(*
Nazwa:			P08_CapFeeder
Opis:			Stacja podajnika nasadek
Wersja:			v0.2
Data:			2024-01-12
Autor:			DP
Urzadzenia:		
Konfiguracja:	
Info:

*)
PROGRAM P08_CapSorter
VAR_INPUT
	IbCapSorterGateScrewerSensor 			:BOOL;			
	IbCapSorterGateWeightSensor				:BOOL;
	//WEJSCIA I WYJSCIA SPRZETOWE
	IbCapSorterDragHomingSensor 			 :BOOL;						// Czujnik bazowania
	QbCapSorterDragActuator               	 :BOOL;						// Siłownikiem przeciągania 
	IbCapSorterDragUpSensor 				 :BOOL;						// Czujnik
	IbCapSorterDragDownSensor 				 :BOOL;						// Czujnik
	                                         
	QbCapSorterDragLeadBefore1Actuator       :BOOL;						// Siłownikiem prowadzenia przed 
	IbCapSorterDragLeadBefore1UpSensor 	 	 :BOOL;						// Czujnik
 	IbCapSorterDragLeadBefore2UpSensor 	 	 :BOOL;						// Czujnik			
	QbCapSorterDragLeadAfter1Actuator        :BOOL;						// Siłownikiem prowadzenia za
	IbCapSorterDragLeadAfter1UpSensor 	 	 :BOOL;						// Czujnik
 	IbCapSorterDragLeadAfter2UpSensor 	 	 :BOOL;						// Czujnik			

END_VAR
VAR
	
	(*******PRZECIAGANIE**********)
	eCapSorterDragStation						: E_Station;
	eCapSorterDragRunningStation				: E_DragStationState;
	fbCapSorterDragState						: FB_State;
	fbCapSorterDragStation						: FB_FormsDragStepper;	
	
	

	
	
	//Pomocnicze
	tofCapSorterDragEnable					: TOF;
	
	//Stoper
	QbCapSorterStoperActuator				: BOOL;				// bit to wysterowania sygnału stopera	
	tpStoperTimerOn							: TP;				// timer do generowania impulsu
	fbStoperSensorDelay						: FB_InputFilter;	// filtr do generowania sygnału 
	lrCapSorterStoperPosition						: LREAL;	
	rtCapSorterStoperDraging: R_TRIG;
	rtCapSorterStoperEndingOfDraging: R_TRIG;	
	//Inne
	bTemp: BOOL;

	rtCapSorterStoperPackMLStarting: R_TRIG;
	bCapSorterStoperWaitingForSensor: BOOL;
	bCapSorterStoperActuatorDelay: BOOL;
	tonbCapSorterStoperActuatorDelay: TON;
	
	//ManualStoper
	rtManualMode	: R_TRIG;
	ftManualMode	: F_TRIG;	
	bCapSorterStoperActuatorLastState	:BOOL;
	
END_VAR

//bCapSorterDisable:=VIS.bCapPuttedCheckIgnoreErrors;


tofCapSorterDragEnable(IN:= GVL.bCapSorterDragEnable, PT:= T#5S);
aLimits();
aStoper();
aDragStation();
aCapSorterWarnings();


(********* GENEROWANIE STANU STACJI DO WIZKI**********)
fbCapSorterDragState(
	eState:=eCapSorterDragStation, 
	bRun:=VIS.bCapSorterDragRun,
	eFormsDragingRunningState:=eCapSorterDragRunningStation, 
	sStateDesc=> VIS.sCapSorterDragState,
	iState=>VIS.iCapSorterDragState);
(***** KONIEC GENEROWANIE STANU STACJI DO WIZKI*******)



IF fbCapSorterDragStation.bCycleDone AND bManualMode THEN
	VIS.bCapSorterDragRun 						:= FALSE;
	GVL.bCapSorterDragPrepareRun				:= FALSE;
END_IF

ACTION aCapSorterWarnings:

//Warning 0
IF stCapSorterRead.eReservedSignals.iReserved20.0 AND NOT CapSorterWarning[0].bWarning THEN
	CapSorterWarning[0].bWarning										:=TRUE;
	CapSorterWarning[0].udiWarningCode									:=41;
	CapSorterWarning[0].sDescription									:='Sorter nasadek | Brak nasadek w zasobniku';
ELSIF NOT stCapSorterRead.eReservedSignals.iReserved20.0 THEN//AND CapSorterWarning[0].bAcknowledge THEN
	CapSorterWarning[0].bWarning										:=FALSE;
	CapSorterWarning[0].bAcknowledge									:=FALSE;
	VIS.uliWarningAcknowledge.27										:=FALSE;
ELSIF CapSorterWarning[0].bAcknowledge THEN                               
	CapSorterWarning[0].bAcknowledge									:=TRUE;
END_IF

//Warning 1
IF stCapSorterRead.eReservedSignals.iReserved20.1 AND NOT CapSorterWarning[1].bWarning THEN
	CapSorterWarning[1].bWarning										:=TRUE;
	CapSorterWarning[1].udiWarningCode									:=42;
	CapSorterWarning[1].sDescription									:='Sorter nasadek | Brak nasadek na stole - sprawdź transporter pośredni';
ELSIF NOT stCapSorterRead.eReservedSignals.iReserved20.1 AND CapSorterWarning[1].bAcknowledge THEN
	CapSorterWarning[1].bWarning										:=FALSE;
	CapSorterWarning[1].bAcknowledge									:=FALSE;
	VIS.uliWarningAcknowledge.28										:=FALSE;
ELSIF CapSorterWarning[1].bAcknowledge THEN
	CapSorterWarning[1].bAcknowledge									:=TRUE;
END_IF

//Warning 2
IF stCapSorterRead.eReservedSignals.iReserved20.2 AND NOT CapSorterWarning[2].bWarning THEN
	CapSorterWarning[2].bWarning										:=TRUE;
	CapSorterWarning[2].udiWarningCode									:=43;
	CapSorterWarning[2].sDescription									:='Sorter nasadek | Niepobrana nasadka przez chwytak 1';
ELSIF NOT stCapSorterRead.eReservedSignals.iReserved20.1 AND CapSorterWarning[2].bAcknowledge THEN
	CapSorterWarning[2].bWarning										:=FALSE;
	CapSorterWarning[2].bAcknowledge									:=FALSE;
	VIS.uliWarningAcknowledge.29										:=FALSE;
ELSIF CapSorterWarning[2].bAcknowledge THEN
	CapSorterWarning[2].bAcknowledge									:=TRUE;
END_IF

//Warning 3
IF stCapSorterRead.eReservedSignals.iReserved20.3 AND NOT CapSorterWarning[3].bWarning THEN
	CapSorterWarning[3].bWarning										:=TRUE;
	CapSorterWarning[3].udiWarningCode									:=44;
	CapSorterWarning[3].sDescription									:='Sorter nasadek | Niepobrana nasadka przez chwytak 2';
ELSIF NOT stCapSorterRead.eReservedSignals.iReserved20.1 AND CapSorterWarning[3].bAcknowledge THEN
	CapSorterWarning[3].bWarning										:=FALSE;
	CapSorterWarning[3].bAcknowledge									:=FALSE;
	VIS.uliWarningAcknowledge.30										:=FALSE;
ELSIF CapSorterWarning[3].bAcknowledge THEN
	CapSorterWarning[3].bAcknowledge									:=TRUE;
END_IF

//Warning 4
IF stCapSorterRead.eReservedSignals.iReserved20.4 AND NOT CapSorterWarning[4].bWarning THEN
	CapSorterWarning[4].bWarning										:=TRUE;
	CapSorterWarning[4].udiWarningCode									:=45;
	CapSorterWarning[4].sDescription									:='Sorter nasadek | Niepobrana nasadka przez chwytak 3';
ELSIF NOT stCapSorterRead.eReservedSignals.iReserved20.1 AND CapSorterWarning[4].bAcknowledge THEN
	CapSorterWarning[4].bWarning										:=FALSE;
	CapSorterWarning[4].bAcknowledge									:=FALSE;
	VIS.uliWarningAcknowledge.31										:=FALSE;
ELSIF CapSorterWarning[4].bAcknowledge THEN
	CapSorterWarning[4].bAcknowledge									:=TRUE;
END_IF

//Warning 5
IF stCapSorterRead.eReservedSignals.iReserved20.5 AND NOT CapSorterWarning[5].bWarning THEN
	CapSorterWarning[5].bWarning										:=TRUE;
	CapSorterWarning[5].udiWarningCode									:=46;
	CapSorterWarning[5].sDescription									:='Sorter nasadek | Niepobrana nasadka przez chwytak 4';	
ELSIF NOT stCapSorterRead.eReservedSignals.iReserved20.1 AND CapSorterWarning[5].bAcknowledge THEN
	CapSorterWarning[5].bWarning										:=FALSE;
	CapSorterWarning[5].bAcknowledge									:=FALSE;
	VIS.uliWarningAcknowledge.32										:=FALSE;
ELSIF CapSorterWarning[5].bAcknowledge THEN
	CapSorterWarning[5].bAcknowledge									:=TRUE;
END_IF
END_ACTION

ACTION aDragStation:
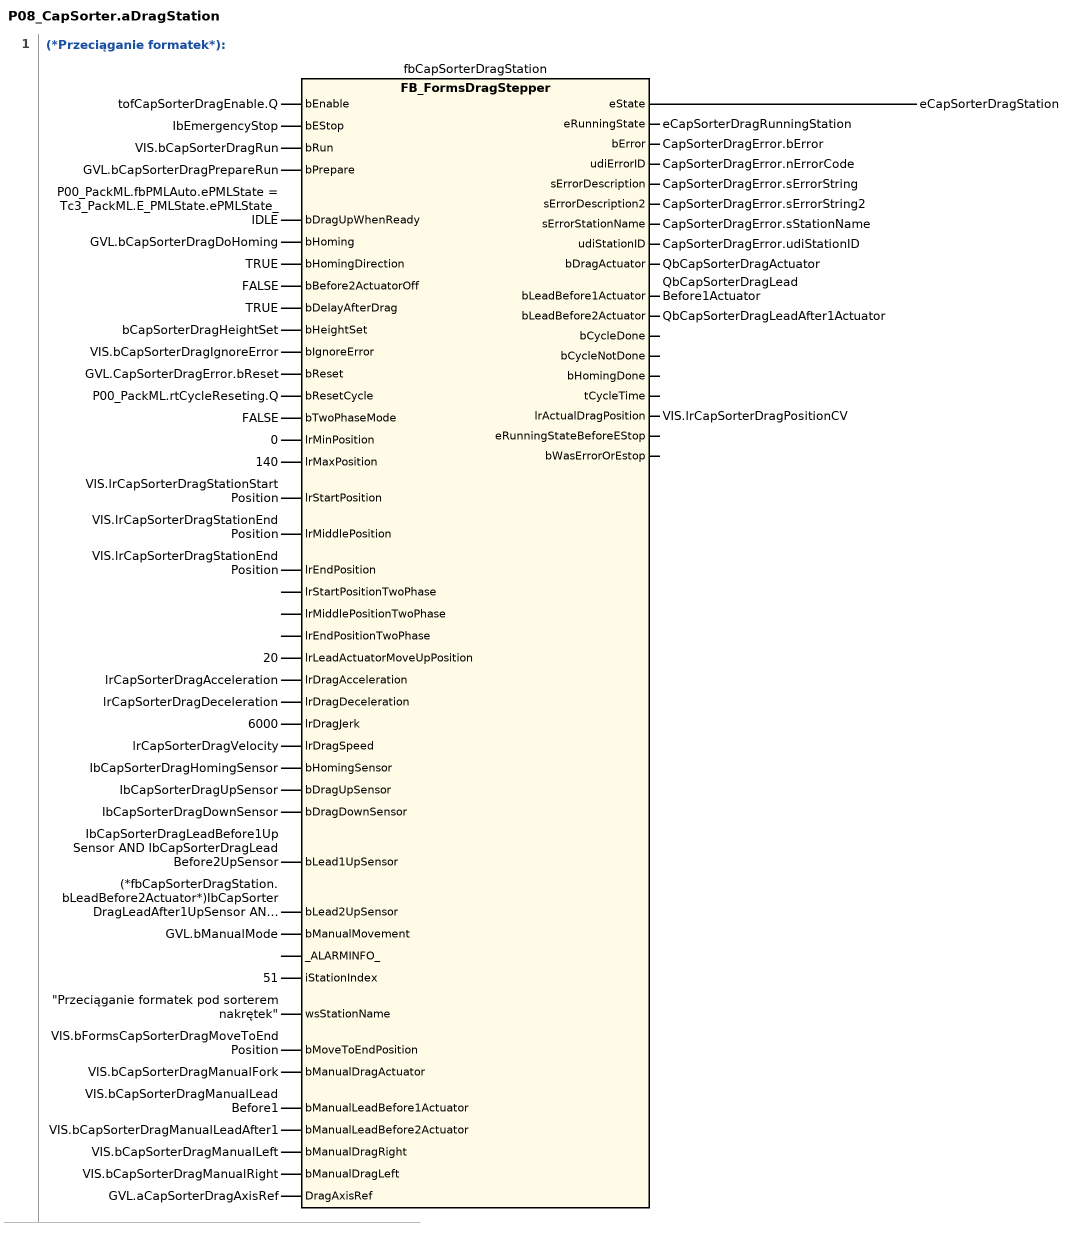
// NETWORK 1
// label: (*Przeciąganie formatek*)
fbCapSorterDragStation(
    bEnable := tofCapSorterDragEnable.Q,
    bEStop := IbEmergencyStop,
    bRun := VIS.bCapSorterDragRun,
    bPrepare := GVL.bCapSorterDragPrepareRun,
    bDragUpWhenReady := P00_PackML.fbPMLAuto.ePMLState = Tc3_PackML.E_PMLState.ePMLState_IDLE,
    bHoming := GVL.bCapSorterDragDoHoming,
    bHomingDirection := TRUE,
    bBefore2ActuatorOff := FALSE,
    bDelayAfterDrag := TRUE,
    bHeightSet := bCapSorterDragHeightSet,
    bIgnoreError := VIS.bCapSorterDragIgnoreError,
    bReset := GVL.CapSorterDragError.bReset,
    bResetCycle := P00_PackML.rtCycleReseting.Q,
    bTwoPhaseMode := FALSE,
    lrMinPosition := 0,
    lrMaxPosition := 140,
    lrStartPosition := VIS.lrCapSorterDragStationStartPosition,
    lrMiddlePosition := VIS.lrCapSorterDragStationEndPosition,
    lrEndPosition := VIS.lrCapSorterDragStationEndPosition,
    lrLeadActuatorMoveUpPosition := 20,
    lrDragAcceleration := lrCapSorterDragAcceleration,
    lrDragDeceleration := lrCapSorterDragDeceleration,
    lrDragJerk := 6000,
    lrDragSpeed := lrCapSorterDragVelocity,
    bHomingSensor := IbCapSorterDragHomingSensor,
    bDragUpSensor := IbCapSorterDragUpSensor,
    bDragDownSensor := IbCapSorterDragDownSensor,
    bLead1UpSensor := IbCapSorterDragLeadBefore1UpSensor AND IbCapSorterDragLeadBefore2UpSensor,
    bLead2UpSensor := (*fbCapSorterDragStation.bLeadBefore2Actuator*)IbCapSorterDragLeadAfter1UpSensor AND IbCapSorterDragLeadAfter2UpSensor,
    bManualMovement := GVL.bManualMode,
    iStationIndex := 51,
    wsStationName := "Przeciąganie formatek pod sorterem nakrętek",
    bMoveToEndPosition := VIS.bFormsCapSorterDragMoveToEndPosition,
    bManualDragActuator := VIS.bCapSorterDragManualFork,
    bManualLeadBefore1Actuator := VIS.bCapSorterDragManualLeadBefore1,
    bManualLeadBefore2Actuator := VIS.bCapSorterDragManualLeadAfter1,
    bManualDragRight := VIS.bCapSorterDragManualLeft,
    bManualDragLeft := VIS.bCapSorterDragManualRight,
    DragAxisRef := GVL.aCapSorterDragAxisRef,
    eRunningState => eCapSorterDragRunningStation,
    bError => CapSorterDragError.bError,
    udiErrorID => CapSorterDragError.nErrorCode,
    sErrorDescription => CapSorterDragError.sErrorString,
    sErrorDescription2 => CapSorterDragError.sErrorString2,
    sErrorStationName => CapSorterDragError.sStationName,
    udiStationID => CapSorterDragError.udiStationID,
    bDragActuator => QbCapSorterDragActuator,
    bLeadBefore1Actuator => QbCapSorterDragLeadBefore1Actuator,
    bLeadBefore2Actuator => QbCapSorterDragLeadAfter1Actuator,
    lrActualDragPosition => VIS.lrCapSorterDragPositionCV); // FB_FormsDragStepper
eCapSorterDragStation := fbCapSorterDragStation.eState;
END_ACTION

ACTION aLimits:
//
IF 	VIS.lrCapSorterDragStationStartPosition		= 0		THEN	VIS.lrCapSorterDragStationStartPosition	:=	7;		END_IF;
IF 	VIS.lrCapSorterDragStationEndPosition		= 0		THEN	VIS.lrCapSorterDragStationEndPosition		:=	142;	END_IF;
END_ACTION

ACTION aStoper:
(*
Nazwa:			aStoper
Opis:			Stoper spowalniania formatek
Wersja:			v0.1
Data:			2024-03-21
Autor:			DP
Urzadzenia:		
Konfiguracja:	
Info:

*)


// 0 - Przliczanie od predkości przeciagania				   
lrCapSorterStoperPosition	 :=	(188.25 * EXPT(lrCapSorterDragVelocity,-0.404));
	

// 1 - Wysuwanie stopera na koniec przesuwania gdy pracuje
rtCapSorterStoperDraging(CLK:=  
								P08_CapSorter.fbCapSorterDragStation.eRunningState = E_DragStationState.eDraging AND 
								((P00_PackML.fbPMLAuto.ePMLState = E_PMLState.ePMLState_STOPPING) OR  (P00_PackML.fbPMLAuto.ePMLState = E_PMLState.ePMLState_EXECUTE)) AND
						   		P08_CapSorter.fbCapSorterDragStation.lrActualDragPosition > lrCapSorterStoperPosition+20 
						,Q=>);
						
IF rtCapSorterStoperDraging.Q THEN
	QbCapSorterStoperActuator	:= TRUE;
END_IF


									
// 2 - Sygnał czekania na czujnik formatek
rtCapSorterStoperPackMLStarting (CLK:=  	
											(P00_PackML.fbPMLAuto.ePMLState = E_PMLState.ePMLState_STARTING)
								,Q=>);

								

//rtCapSorterStoperEndingOfDraging(CLK:=  	P08_CapSorter.fbCapSorterDragStation.eRunningState = E_DragStationState.eDraged AND 
rtCapSorterStoperEndingOfDraging(CLK:=  	P08_CapSorter.fbCapSorterDragStation.eRunningState = E_DragStationState.eDragingDone AND 
											((P00_PackML.fbPMLAuto.ePMLState = E_PMLState.ePMLState_STOPPING) OR  (P00_PackML.fbPMLAuto.ePMLState = E_PMLState.ePMLState_EXECUTE))
								,Q=>);
						

IF rtCapSorterStoperEndingOfDraging.Q OR rtCapSorterStoperPackMLStarting.Q THEN
	bCapSorterStoperWaitingForSensor	:=	TRUE;	
END_IF							

// 3 - Wyłączanie stopera
IF NOT bDosingTwoPhases THEN
	IF bCapSorterStoperWaitingForSensor AND P00_PackML.fbIbCapSorterFourthFormCheckFormSensor.bOut THEN	
		bCapSorterStoperActuatorDelay	:=	TRUE;
	END_IF
ELSE
	IF bCapSorterStoperWaitingForSensor (*AND MAIN.IbCapSorterFourthFormCheckFormSensor*) AND iCapSorterDragFormCounter >=1 AND P00_ReadRFIDCard.bReadedCardCapSorter THEN	
		bCapSorterStoperActuatorDelay	:=	TRUE;
	END_IF
END_IF

IF 	nFormTransportersBeforeScrewerVelocitySV < 610 AND NOT bDosingTwoPhases THEN
	tonbCapSorterStoperActuatorDelay(IN:=bCapSorterStoperActuatorDelay, PT:=T#1S150MS);
ELSE
	tonbCapSorterStoperActuatorDelay(IN:=bCapSorterStoperActuatorDelay, PT:=T#790MS);//990
END_IF

IF tonbCapSorterStoperActuatorDelay.Q THEN
	bCapSorterStoperActuatorDelay		:=	FALSE;
	bCapSorterStoperWaitingForSensor	:=	FALSE;
	QbCapSorterStoperActuator			:=	FALSE;
END_IF


//Manual
rtManualMode	(CLK:=bManualMode,	Q=>);
ftManualMode	(CLK:=bManualMode,	Q=>);
IF rtManualMode.Q THEN
	bCapSorterStoperActuatorLastState	:=	QbCapSorterStoperActuator;
	VIS.bCapSorterStoperManualActuator	:=	QbCapSorterStoperActuator;
END_IF
IF bManualMode THEN
	QbCapSorterStoperActuator			:=	VIS.bCapSorterStoperManualActuator;
END_IF
IF ftManualMode.Q THEN
	QbCapSorterStoperActuator			:= bCapSorterStoperActuatorLastState;
END_IF
// Koniec Manual
END_ACTION

END_PROGRAM

(* stored: Version 1.1.0.1, ProductVersion 3.1.4026.13, FileIdentifier 95ae5d9537bb561c0f398f819fc31a04e94d9eb2, FileSignature 778299434e2d21aa2116f38940a754af116e279265ab9f7386e0e01eda16ae888085d10aa1a9ee26267131437cae21ec81cb56072cbcfb2701091d909d2f55781187718e969c6a0c2bb548f8dd39127fab1cb5a28712a4bf10fc53b53bb772f3f3321a84706a1938af7910d8b6dc704872ffca7d6c7ee7a44a7b66b7ee8452fb42cf5497c990f3daf32b8efdbdcd2ccc9e3651de323bbde93241559fb336d9eb2d94404a61bbc229e69e475ede6b5ec6a7bcb36370055ea372259c577266d239bb8922affbb9d8633a9462c68c6920a443cfaee4786d33ace3a96538351d5f77d786f53d743424eb4ef429366502bc2a12fabdbd9bdedbd4fdc8ce7fc41d6498
   POU P08_CapSorter: Id {d4ffcb5b-9c49-4962-b941-b9f7d2070f0b}, SpecialFunc None
   Action aCapSorterWarnings: Id {9b30c933-17a4-4719-b144-820fb6c68a68}
   Action aDragStation: Id {7aed2a45-0fdf-410d-a07e-0cfa3dcb8435}
   Action aLimits: Id {7b3d5216-fb15-489d-82a1-a55ffb8945bf}
   Action aStoper: Id {5cae9897-2fa2-4a7f-b548-09a6cbd6f35a} *)
